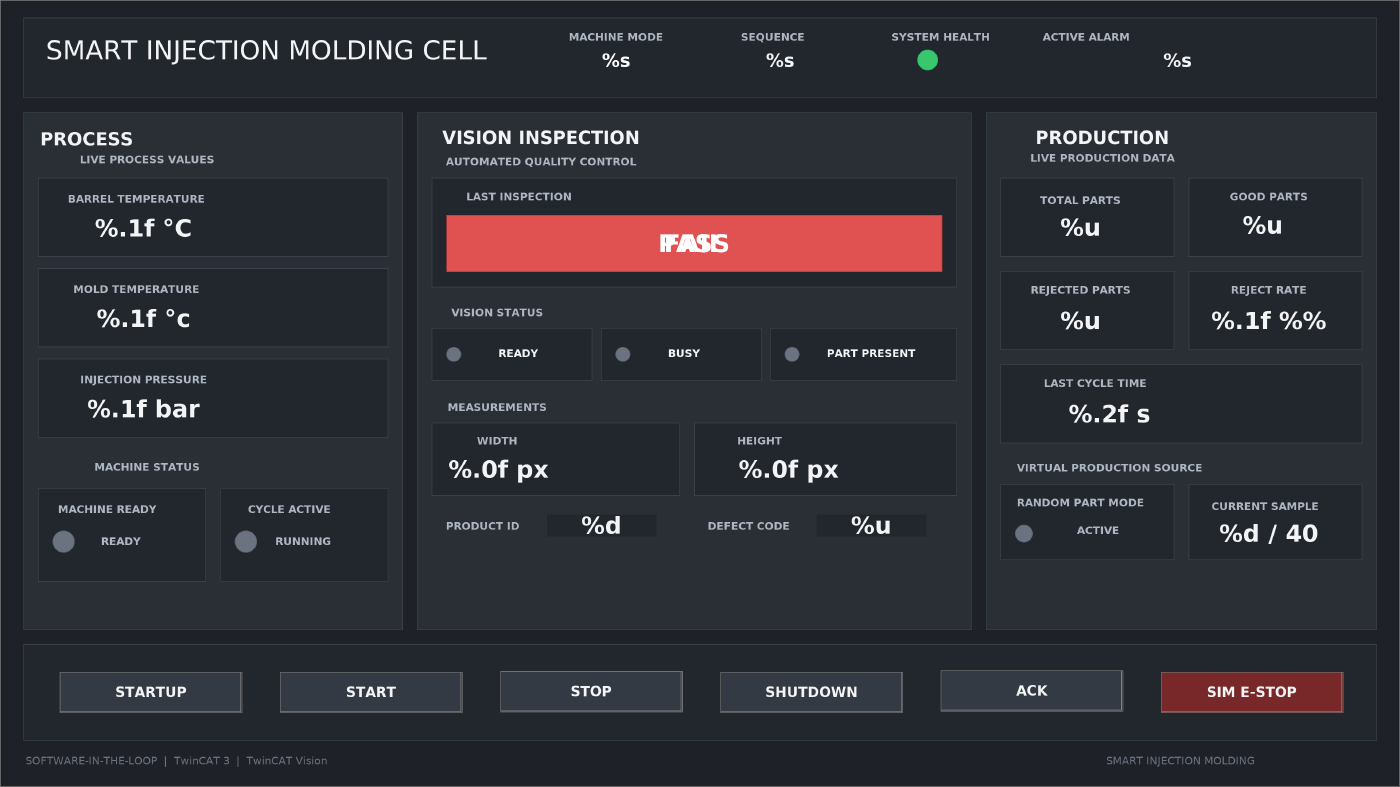
VISUALIZATION Visualization_Overview  // 1920x1080
    Rectangle (32,24 1856x110)
    Rectangle (32,154 520x710)
    Rectangle (572,154 760x710)
    Rectangle (1352,154 536x710)
    Rectangle (32,884 1856x132)
    Label (60,48 747x42), "SMART INJECTION MOLDING CELL"
    Label (760,41 170x20), "MACHINE MODE"
    Textfield (760,66 170x34), "%s", text variable: GVL_Status.sMachineModeText
    Label (960,41 210x20), "SEQUENCE"
    Textfield (960,66 220x34), "%s", text variable: GVL_Status.sSequenceText
    Label (1210,41 160x20), "SYSTEM HEALTH"
    Ellipse (1258,68 28x28), colour toggle: GVL_Status.bFaultActive
    Label (1400,41 180x20), "ACTIVE ALARM"
    Textfield (1400,66 430x34), "%s", text variable: GVL_Status.sActiveAlarmText
    Button (82,922 250x56), "STARTUP", colour toggle: GVL_IO.B_startup
        tap GVL_IO.B_startup
    Button (384,922 250x56), "START", colour toggle: GVL_IO.B_start
        tap GVL_IO.B_start
    Button (686,921 250x56), "STOP", colour toggle: GVL_IO.B_stop
        tap GVL_IO.B_stop
    Button (988,922 250x56), "SHUTDOWN", colour toggle: GVL_IO.B_shutdown
        tap GVL_IO.B_shutdown
    Button (1290,920 250x56), "ACK", colour toggle: GVL_IO.B_ack
        tap GVL_IO.B_ack
    Button (1592,922 250x56), "SIM E-STOP", colour toggle: GVL_IO.B_ES
        toggle GVL_IO.B_ES
    Label (52,174 300x34), "PROCESS"
    Label (52,208 300x22), "LIVE PROCESS VALUES"
    Rectangle (52,244 480x108)
    Label (72,262 230x22), "BARREL TEMPERATURE"
    Textfield (72,292 250x42), "%.1f °C", text variable: GVL_Status.fBarrelTemp
    Rectangle (52,368 480x108)
    Label (72,386 230x22), "MOLD TEMPERATURE"
    Textfield (72,416 250x42), "%.1f °c", text variable: GVL_Status.fMoldTemp
    Rectangle (52,492 480x108)
    Label (72,510 250x22), "INJECTION PRESSURE"
    Textfield (72,540 250x42), "%.1f bar", text variable: GVL_Status.fPressureBar
    Label (52,628 300x26), "MACHINE STATUS"
    Rectangle (52,670 230x128)
    Label (72,688 150x22), "MACHINE READY"
    Ellipse (72,728 30x30), colour toggle: GVL_Status.bMachineReady
    Label (116,730 100x26), "READY"
    Rectangle (302,670 230x128)
    Label (322,688 150x22), "CYCLE ACTIVE"
    Ellipse (322,728 30x30), colour toggle: GVL_Status.bCycleActive
    Label (366,730 100x26), "RUNNING"
    Label (592,174 300x30), "VISION INSPECTION"
    Label (592,207 300x30), "AUTOMATED QUALITY CONTROL"
    Rectangle (592,244 720x150)
    Label (612,260 200x20), "LAST INSPECTION"
    Rectangle (612,295 680x78), colour toggle: GVL_Status.stVision.bPartOK
    Label (612,295 680x78), "PASS", invisible if: NOT GVL_Status.stVision.bPartOK
    Label (612,295 680x78), "FAIL", invisible if: GVL_Status.stVision.bPartOK
    Label (592,418 180x22), "VISION STATUS"
    Rectangle (592,450 220x72)
    Ellipse (612,476 20x20), colour toggle: GVL_Status.stVision.bReady
    Label (646,470 130x30), "READY"
    Rectangle (824,450 220x72)
    Ellipse (844,476 20x20), colour toggle: GVL_Status.stVision.bBusy
    Label (878,470 120x30), "BUSY"
    Rectangle (1056,450 256x72)
    Label (1110,470 170x30), "PART PRESENT"
    Ellipse (1076,476 20x20), colour toggle: GVL_Status.stVision.bPartPresent
    Label (592,548 180x22), "MEASUREMENTS"
    Rectangle (592,580 340x100)
    Label (612,595 140x20), "WIDTH"
    Textfield (612,625 220x38), "%.0f px", text variable: GVL_Status.stVision.fWidth
    Rectangle (952,580 360x100)
    Label (972,595 140x20), "HEIGHT"
    Textfield (972,625 220x38), "%.0f px", text variable: GVL_Status.stVision.fHeight
    Label (592,710 140x24), "PRODUCT ID"
    Textfield (750,706 150x30), "%d", text variable: GVL_Status.stVision.nProductID
    Label (952,710 160x24), "DEFECT CODE"
    Textfield (1120,706 150x30), "%u", text variable: GVL_Status.stVision.nDefectCode
    Label (1372,174 280x30), "PRODUCTION"
    Label (1372,207 280x20), "LIVE PRODUCTION DATA"
    Rectangle (1372,244 238x108)
    Label (1392,260 180x30), "TOTAL PARTS"
    Textfield (1392,291 180x42), "%u", text variable: GVL_Status.stProduction.nTotalParts
    Label (1642,257 180x30), "TOTAL PARTS"
    Rectangle (1630,244 238x108)
    Textfield (1642,288 180x42), "%u", text variable: GVL_Status.stProduction.nGoodParts
    Label (1391,398 180x30), "TOTAL PARTS"
    Rectangle (1372,372 238x108)
    Textfield (1392,419 180x42), "%u", text variable: GVL_Status.stProduction.nRejectedParts
    Label (1644,401 180x30), "TOTAL PARTS"
    Rectangle (1630,372 238x108)
    Textfield (1650,419 180x42), "%.1f %%", text variable: GVL_Status.stProduction.fRejectRate
    Label (1396,724 180x30), "TOTAL PARTS"
    Rectangle (1372,664 238x104)
    Label (1650,260 180x20), "GOOD PARTS"
    Rectangle (1630,664 238x104)
    Textfield (1650,714 180x36), "%d / 40", text variable: GVL_Simulation.nVisionDatasetIndex
    Label (1392,388 180x20), "REJECTED PARTS"
    Label (1650,388 180x20), "REJECT RATE"
    Label (1392,680 180x20), "RANDOM PART MODE"
    Label (1650,680 170x30), "CURRENT SAMPLE"
    Rectangle (1372,500 496x108)
    Label (1392,516 220x20), "LAST CYCLE TIME"
    Textfield (1392,547 260x42), "%.2f s", text variable: GVL_Status.stProduction.fLastCycleTimeSec
    Label (1372,632 300x20), "VIRTUAL PRODUCTION SOURCE"
    Ellipse (1392,720 24x24), colour toggle: GVL_Simulation.bRandomPartMode
    Label (1431,713 150x30), "ACTIVE"
    Label (32,1034 900x20), "SOFTWARE-IN-THE-LOOP | TwinCAT 3 | TwinCAT Vision"
    Label (1350,1034 538x20), "SMART INJECTION MOLDING"
END_VISUALIZATION

(* stored: Version 1.1.0.1, ProductVersion 3.1.4024.16
   Visu Visualization_Overview: Id {fd1de266-cf8f-4c39-9e1d-2be1c9891768} *)
